FUNCTION_BLOCK ABSTRACT FBA_TrifectaDrive EXTENDS FBA_Drive
VAR //constructor
	enableDualSideTraverse : BOOL;
END_VAR
VAR
	outerLimit AT %I* : BOOL;
END_VAR
(*
this abstract FB adds a rear limit sensor to FBA_Drive
*)

{attribute 'monitoring':='call'}
PROPERTY AtOuterLimit : BOOL
GET
AtOuterLimit := outerLimit <> limitSensorDefaultState;
END_GET
END_PROPERTY

END_FUNCTION_BLOCK

(* stored: Version 1.1.0.1, ProductVersion 3.1.4024.11
   POU FBA_TrifectaDrive: Id {f410d910-3fd9-42f5-8bfc-6a2906d78af5}, SpecialFunc None
   Property AtOuterLimit: Id {e02ad79c-ff8f-4672-8eae-eab46f608664}
   Get Get: Id {3e341a5b-d3a7-4ac5-beec-589afe8ba200} *)
